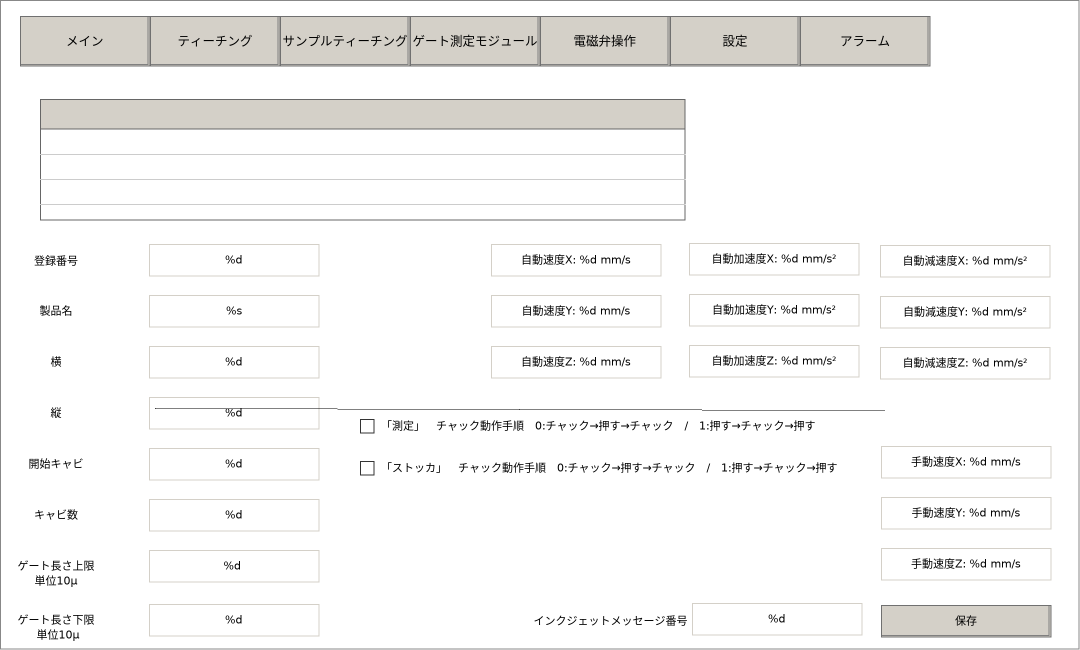
VISUALIZATION s_addNewProduct  // 1080x650
    Rectangle (0,0 1080x650)
    Textfield (149,346 170x32), "%d", text variable: gvl_visu.var_in_productGenerate.bottomPocketQty
        OnMouseClick: write gvl_visu.var_in_productGenerate.bottomPocketQty via VisuDialogs.Numpad
    Textfield (149,397 170x32), "%d", text variable: gvl_visu.var_in_productGenerate.vertivalPocketQty
        OnMouseClick: write gvl_visu.var_in_productGenerate.vertivalPocketQty via VisuDialogs.Numpad
    Textfield (149,499 170x32), "%d", text variable: gvl_visu.var_in_productGenerate.cavQty
        OnMouseClick: write gvl_visu.var_in_productGenerate.cavQty via VisuDialogs.Numpad
    Textfield (149,448 170x32), "%d", text variable: gvl_visu.var_in_productGenerate.startCav
        OnMouseClick: write gvl_visu.var_in_productGenerate.startCav via VisuDialogs.Numpad
    Label (6,398 100x30), "縦"
    Label (6,347 100x30), "横"
    Label (6,500 100x30), "キャビ数"
    Label (6,449 100x30), "開始キャビ"
    Textfield (149,295 170x32), "%s", text variable: gvl_visu.var_in_productGenerate.name
        OnMouseClick: write gvl_visu.var_in_productGenerate.name via VisuDialogs.Keypad
    Label (6,296 100x30), "製品名"
    Label (6,246 100x30), "登録番号"
    Textfield (149,244 170x32), "%d", text variable: gvl_visu.var_in_productGenerate.num
        OnMouseClick: write gvl_visu.var_in_productGenerate.num via VisuDialogs.Numpad
    Textfield (149,550 170x32), "%d", text variable: gvl_visu.var_in_productGenerate.gateLength_max
        OnMouseClick: write gvl_visu.var_in_productGenerate.gateLength_max via VisuDialogs.Numpad
    Label (6,551 100x30), "ゲート長さ上限"
    Label (6,605 100x30), "ゲート長さ下限"
    Table (40,99 645x121), data array: gvl_param.var_productInfo
        p3854506369: gvl_param.var_productInfo[INDEX].num
        p1892666644: gvl_param.var_productInfo[INDEX].name
        p338671338: gvl_param.var_productInfo[INDEX].cavQty
        p2170511999: gvl_param.var_productInfo[INDEX].bottomPocketQty
        p3723444502: gvl_param.var_productInfo[INDEX].vertivalPocketQty
        p1218418051: gvl_param.var_productInfo[INDEX].pocketSumQty
        p746581629: gvl_param.var_productInfo[INDEX].startCav
        p3104783080: gvl_param.var_productInfo[INDEX].gateLength_min
        p2501879983: gvl_param.var_productInfo[INDEX].gateLength_max
        p2232123230: 番号
        p511219082: 製品名
        p1755163831: キャビ数
        p4092479075: トレイ横数
        p2237128397: トレイ縦数
        p505689113: 入り数
        p1757482276: 開始キャビ
        p4088588272: ゲート下限
        p2243050616: ゲート上限
        p7306298: gvl_param.var_productInfo[INDEX].teachPos
        p1933151965: gvl_param.var_productInfo[INDEX].autoVels
        p3863566920: gvl_param.var_productInfo[INDEX].manaulVels
    Textfield (149,604 170x32), "%d", text variable: gvl_visu.var_in_productGenerate.gateLength_min
        OnMouseClick: write gvl_visu.var_in_productGenerate.gateLength_min via VisuDialogs.Numpad
    Textfield (491,295 170x32), "自動速度Y: %d mm/s", text variable: gvl_visu.var_in_productGenerate.autoVels.y.vel
        OnMouseClick: write gvl_visu.var_in_productGenerate.autoVels.y.vel via VisuDialogs.Numpad
    Textfield (491,346 170x32), "自動速度Z: %d mm/s", text variable: gvl_visu.var_in_productGenerate.autoVels.z.vel
        OnMouseClick: write gvl_visu.var_in_productGenerate.autoVels.z.vel via VisuDialogs.Numpad
    Textfield (881,497 170x32), "手動速度Y: %d mm/s", text variable: gvl_visu.var_in_productGenerate.manaulVels.y.vel
        OnMouseClick: write gvl_visu.var_in_productGenerate.manaulVels.y.vel via VisuDialogs.Numpad
    Textfield (881,446 170x32), "手動速度X: %d mm/s", text variable: gvl_visu.var_in_productGenerate.manaulVels.x.vel
        OnMouseClick: write gvl_visu.var_in_productGenerate.manaulVels.x.vel via VisuDialogs.Numpad
    Textfield (491,244 170x32), "自動速度X: %d mm/s", text variable: gvl_visu.var_in_productGenerate.autoVels.x.vel
        OnMouseClick: write gvl_visu.var_in_productGenerate.autoVels.x.vel via VisuDialogs.Numpad
    Textfield (881,548 170x32), "手動速度Z: %d mm/s", text variable: gvl_visu.var_in_productGenerate.manaulVels.z.vel
        OnMouseClick: write gvl_visu.var_in_productGenerate.manaulVels.z.vel via VisuDialogs.Numpad
    Button (881,605 170x32), "保存"
        tap gvl_visu.flg_btn_saveProductInfo
    Textfield (689,294 170x32), "自動加速度Y: %d mm/s²", text variable: gvl_visu.var_in_productGenerate.autoVels.y.acc
        OnMouseClick: write gvl_visu.var_in_productGenerate.autoVels.y.acc via VisuDialogs.Numpad
    Textfield (689,345 170x32), "自動加速度Z: %d mm/s²", text variable: gvl_visu.var_in_productGenerate.autoVels.z.acc
        OnMouseClick: write gvl_visu.var_in_productGenerate.autoVels.z.acc via VisuDialogs.Numpad
    Textfield (689,243 170x32), "自動加速度X: %d mm/s²", text variable: gvl_visu.var_in_productGenerate.autoVels.x.acc
        OnMouseClick: write gvl_visu.var_in_productGenerate.autoVels.x.acc via VisuDialogs.Numpad
    Textfield (880,296 170x32), "自動減速度Y: %d mm/s²", text variable: gvl_visu.var_in_productGenerate.autoVels.y.dcc
        OnMouseClick: write gvl_visu.var_in_productGenerate.autoVels.y.dcc via VisuDialogs.Numpad
    Textfield (880,347 170x32), "自動減速度Z: %d mm/s²", text variable: gvl_visu.var_in_productGenerate.autoVels.z.dcc
        OnMouseClick: write gvl_visu.var_in_productGenerate.autoVels.z.dcc via VisuDialogs.Numpad
    Textfield (880,245 170x32), "自動減速度X: %d mm/s²", text variable: gvl_visu.var_in_productGenerate.autoVels.x.dcc
        OnMouseClick: write gvl_visu.var_in_productGenerate.autoVels.x.dcc via VisuDialogs.Numpad
    Line (155,408) (884,410)
    Label (6,566 100x30), "単位10μ"
    Label (8,620 100x30), "単位10μ"
    Textfield (692,603 170x32), "%d", text variable: gvl_visu.var_in_productGenerate.incjetMsgNo
        OnMouseClick: write gvl_visu.var_in_productGenerate.incjetMsgNo via VisuDialogs.Numpad
    Label (537,606 147x30), "インクジェットメッセージ番号"
    Button (20,16 130x50), "メイン"
        OnMouseClick: change screen: s_auto
    Button (150,16 130x50), "ティーチング"
        OnMouseClick: change screen: s_teaching1
    Button (670,16 130x50), "設定"
        OnMouseClick: change screen: s_setting
    Button (540,16 130x50), "電磁弁操作"
        OnMouseClick: change screen: s_manual
    Button (410,16 130x50), "ゲート測定モジュール"
        OnMouseClick: change screen: s_gm_teaching
    Button (800,16 130x50), "アラーム", colour toggle: gvl_io.flg_signalTowerRed
        OnMouseClick: change screen: s_alarm
    Button (280,16 130x50), "サンプルティーチング"
        OnMouseClick: change screen: s_sample
    Checkbox (358,411 505x30), "「測定」 チャック動作手順 0:チャック→押す→チャック / 1:押す→チャック→押す", variable: gvl_visu.var_in_productGenerate.flg_mode_measurement
    Checkbox (358,453 503x30), "「ストッカ」 チャック動作手順 0:チャック→押す→チャック / 1:押す→チャック→押す", variable: gvl_visu.var_in_productGenerate.flg_mode_stocker
END_VISUALIZATION

(* stored: Version 1.1.0.1, ProductVersion 3.1.4024.11
   Visu s_addNewProduct: Id {dd4e99ac-2886-4e75-b4cd-73cedb8c4a7c} *)
